FUNCTION_BLOCK LiftControl (* Basic Function Block Type *)
  (* Standard: 61499-2 *)
  (* Version 0.0, 1/14/2024, midxav, Template *)
  PACKAGE Main;
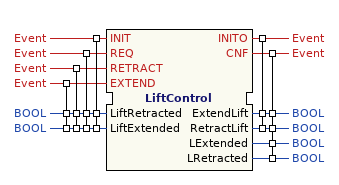
  EVENT_INPUT
    INIT WITH LiftRetracted, LiftExtended; (* Initialization Request *)
    REQ WITH LiftRetracted, LiftExtended; (* Normal Execution Request *)
    RETRACT WITH LiftRetracted, LiftExtended;
    EXTEND WITH LiftRetracted, LiftExtended;
  END_EVENT
  EVENT_OUTPUT
    INITO WITH ExtendLift, RetractLift; (* Initialization Confirm *)
    CNF WITH ExtendLift, RetractLift, LExtended, LRetracted; (* Execution Confirmation *)
  END_EVENT
  VAR_INPUT
    LiftRetracted : BOOL; (* Input event qualifier *)
    LiftExtended : BOOL;
  END_VAR
  VAR_OUTPUT
    ExtendLift : BOOL; (* Output event qualifier *)
    RetractLift : BOOL;
    LExtended : BOOL;
    LRetracted : BOOL;
  END_VAR
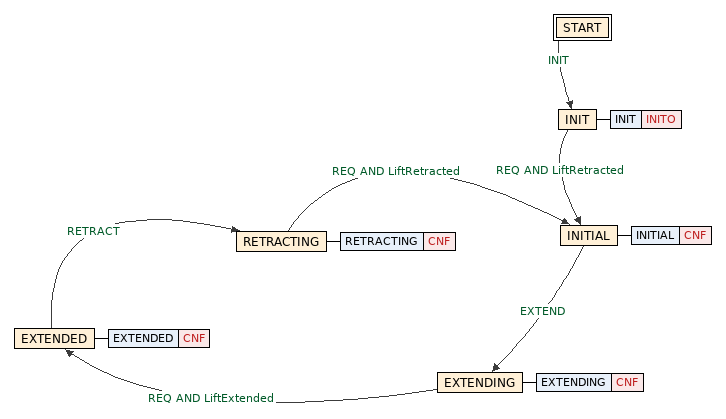
  EC_STATES
    START; (* Initial State *)
    INIT : INIT -> INITO; (* Initialization *)
    INITIAL : INITIAL -> CNF;
    EXTENDING : EXTENDING -> CNF;
    EXTENDED : EXTENDED -> CNF;
    RETRACTING : RETRACTING -> CNF;
  END_STATES
  EC_TRANSITIONS
    START TO INIT := INIT;
    INIT TO INITIAL := REQ AND LiftRetracted;
    INITIAL TO EXTENDING := EXTEND;
    EXTENDING TO EXTENDED := REQ AND LiftExtended;
    EXTENDED TO RETRACTING := RETRACT;
    RETRACTING TO INITIAL := REQ AND LiftRetracted;
  END_TRANSITIONS
  ALGORITHM INIT IN ST:
ExtendLift:= FALSE;
RetractLift:=TRUE;
LExtended:=FALSE;
LRetracted:= FALSE;
  END_ALGORITHM
  ALGORITHM INITIAL IN ST:
RetractLift:=FALSE;
LRetracted := TRUE;
  END_ALGORITHM
  ALGORITHM EXTENDING IN ST:
ExtendLift:=TRUE;
LRetracted:=FALSE;
  END_ALGORITHM
  ALGORITHM EXTENDED IN ST:
ExtendLift:=FALSE;
LExtended :=TRUE;
  END_ALGORITHM
  ALGORITHM RETRACTING IN ST:
RetractLift:=TRUE;
LExtended := FALSE;
  END_ALGORITHM
END_FUNCTION_BLOCK
